// TIA Portal V20 export
DATA_BLOCK "InterfaceTP_C1"   // DB110
// stored: Access Published, MemoryReserve 100
   VAR
      operationOFF : Bool;   // Anlage AUS (HMI) Handbetrieb / operation ON (HMI) manual mode
      operationON : Bool;   // Anlage EIN (HMI) Automatikbetrieb / operation ON (HMI) automatic mode
      jogRight : Bool;   // Bandmotor Tippen Rechts / jog conveyor right
      jogLeft : Bool;   // Bandmotor Tippen Links / jog conveyor left
      acknowledgeFault : Bool;   // Band-Störung quittieren / acknowledge conveyor fault
      actualValue : UInt;   // Ist-Stückzahl / actual value
      setpoint : UInt := 3;   // Sollwert / setpoint value
      operation : Bool;
      conveyorFault : Bool;
   END_VAR
BEGIN
END_DATA_BLOCK
